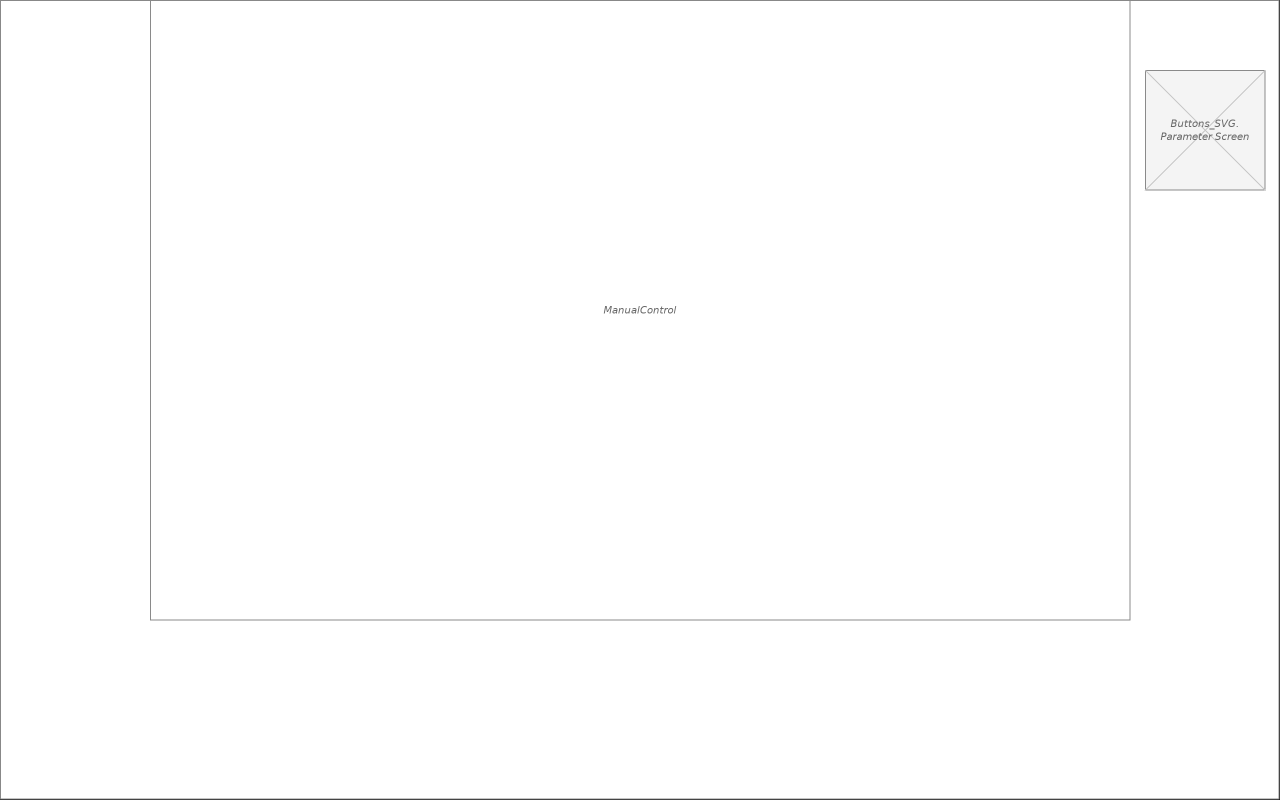
VISUALIZATION Manual  // 1280x800
VAR_IN_OUT
	bCmdParameter : BOOL ;
END_VAR
    Frame (150,0 980x620)
        shows ManualControl()
    Image (1145,70 120x120), image: Buttons_SVG.Parameter Screen
        OnMouseClick: toggle bCmdParameter
    Rectangle (0,0 1280x800)
END_VISUALIZATION

(* stored: Version 1.1.0.1, ProductVersion 3.1.4024.5
   Visu Manual: Id {8b12630b-f7fc-46df-9948-3293bcc3e0af} *)
